SUBAPPLICATION ZaehlerVergleich (* Subapplication Type *)
  (* Standard: 61499-2 *)
  (* Version 1.0, 2023-02-18, Franz *)
  PACKAGE FBs::Counter::subs::Zaehler;
  IMPORT FBs::Counter::const::DefaultPool::OutputString_ZielErreicht;
  IMPORT isobus::UT::Q::const::IDs::ID_NULL;
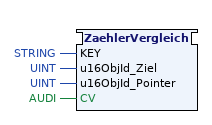
  VAR_INPUT
    KEY : STRING;
    u16ObjId_Ziel : UINT;
    u16ObjId_Pointer : UINT;
  END_VAR
  SOCKETS
    CV : adapter::types::unidirectional::AUDI; (* Counter Value *)
  END_SOCKETS
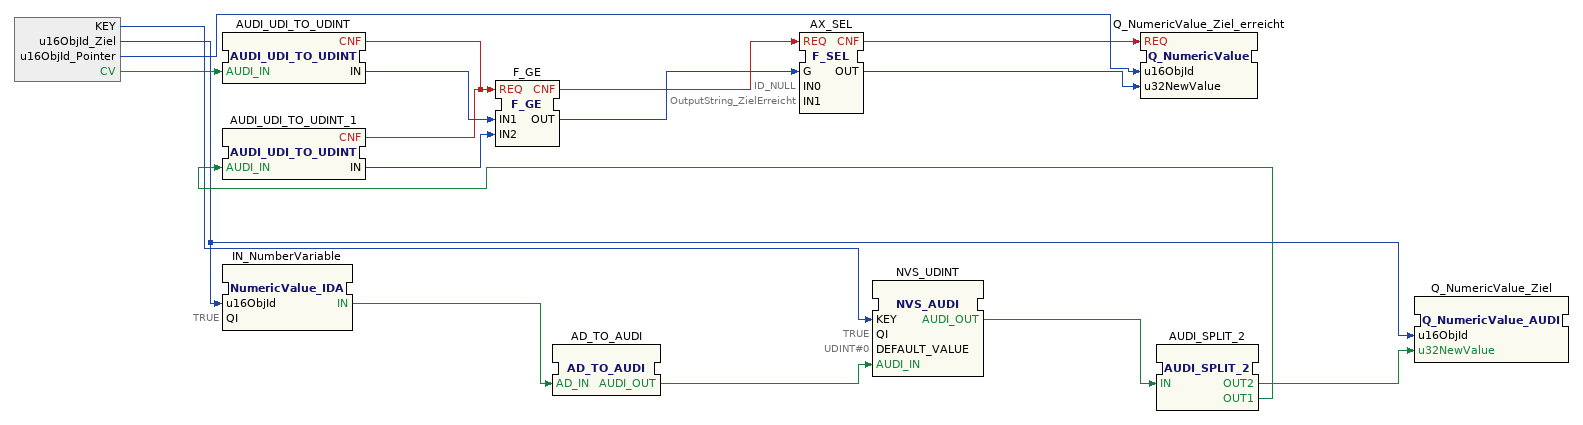
  FBS
    Q_NumericValue_Ziel_erreicht : isobus::UT::Q::Q_NumericValue;
    F_GE : iec61131::comparison::F_GE;
    NVS_UDINT : logiBUS::storage::esp32_nvs::NVS_AUDI(QI := TRUE, DEFAULT_VALUE := UDINT#0);
    Q_NumericValue_Ziel : isobus::UT::Q::Q_NumericValue_AUDI;
    AX_SEL : iec61131::selection::F_SEL(IN0 := ID_NULL, IN1 := OutputString_ZielErreicht);
    IN_NumberVariable : isobus::UT::io::NumericValue::NumericValue_IDA(QI := TRUE);
    AD_TO_AUDI : adapter::conversion::unidirectional::AD_TO_AUDI;
    AUDI_SPLIT_2 : adapter::events::unidirectional::AUDI_SPLIT_2;
    AUDI_UDI_TO_UDINT : adapter::conversion::unidirectional::AUDI_UDI_TO_UDINT;
    AUDI_UDI_TO_UDINT_1 : adapter::conversion::unidirectional::AUDI_UDI_TO_UDINT;
  END_FBS
  EVENT_CONNECTIONS
    AX_SEL.CNF TO Q_NumericValue_Ziel_erreicht.REQ;
    AUDI_UDI_TO_UDINT.CNF TO F_GE.REQ;
    AUDI_UDI_TO_UDINT_1.CNF TO F_GE.REQ;
    F_GE.CNF TO AX_SEL.REQ;
  END_CONNECTIONS
  DATA_CONNECTIONS
    u16ObjId_Pointer TO Q_NumericValue_Ziel_erreicht.u16ObjId;
    AX_SEL.OUT TO Q_NumericValue_Ziel_erreicht.u32NewValue;
    u16ObjId_Ziel TO Q_NumericValue_Ziel.u16ObjId;
    KEY TO NVS_UDINT.KEY;
    u16ObjId_Ziel TO IN_NumberVariable.u16ObjId;
    AUDI_UDI_TO_UDINT.IN TO F_GE.IN1;
    AUDI_UDI_TO_UDINT_1.IN TO F_GE.IN2;
    F_GE.OUT TO AX_SEL.G;
  END_CONNECTIONS
  ADAPTER_CONNECTIONS
    IN_NumberVariable.IN TO AD_TO_AUDI.AD_IN;
    AD_TO_AUDI.AUDI_OUT TO NVS_UDINT.AUDI_IN;
    AUDI_SPLIT_2.OUT2 TO Q_NumericValue_Ziel.u32NewValue;
    NVS_UDINT.AUDI_OUT TO AUDI_SPLIT_2.IN;
    CV TO AUDI_UDI_TO_UDINT.AUDI_IN;
    AUDI_SPLIT_2.OUT1 TO AUDI_UDI_TO_UDINT_1.AUDI_IN;
  END_CONNECTIONS
END_SUBAPPLICATION
